// TIA Portal V17 export
// export: Created 2024-09-02T12:49:55.3240184Z, ExportSetting WithDefaults, DisplayName Totally Integrated Automation Portal, DisplayVersion V17, DisplayName TIA Portal Openness, DisplayVersion V17, DisplayName TIA Portal Version Control Interface, DisplayVersion V17, DisplayName STEP 7 Professional, DisplayVersion V17, DisplayName STEP 7 Safety, DisplayVersion V17, DisplayName WinCC Professional, DisplayVersion V17
FUNCTION "SysFC_AnzTrueDez" : Void   // FC128, LAD
TITLE = Count number of bits with value true / Anzahl Bits mit Wert true zaehlen
{ S7_Optimized_Access := 'TRUE' }
AUTHOR : OlegFuehrus
FAMILY : DIAG
NAME : DIAG
VERSION : 0.1
// stored: AutoNumber true, IsIECCheckEnabled false, SetENOAutomatically false, UDAEnableTagReadback false
   VAR_INPUT
      AnfangBits : Int;   // esrtes Bit zum zaehlen im Array / esrtes bit to count in array
      Anzahl : Int;   // Anzahl Bits zum überprüfen / Number of bits to check
      Daten : Variant;
   END_VAR
   VAR_OUTPUT
      AnzahlTrue : Int;   // Anzahl der Bits mit Wert True / Number of bits with value True
      NrTrue : Int;   // Nummer des ersten gefundenen Bits / Number of the first bit found
   END_VAR
   VAR_TEMP
      t_VKE0 : Bool;
      t_VKE1 : Bool;
      t_RetVal : Word;
      t_AnzahlElemente : UDInt;
      t_AnzahlTrue : Int;
      t_NrTrue : Int;
      t_PosNr : DInt;
      t_UDINT : UDInt;
      t_INT : Int;
      t_Counter : Int;
      t_StartCounter : Int;
      t_EndCounter : Int;
      t_Bool : Bool;
      t_Fehler : Bool;
      t_TypIO : Bool;
      t_DatenByte : Array[1..128] of Byte;
      t_DatenBool : Array[1..1024] of Bool;
   END_VAR
   VAR_TEMP   // added for the SCL form of the ladder/FBD networks
      _w1 : Bool;
   END_VAR
BEGIN

REGION Network 1: VKE0/1
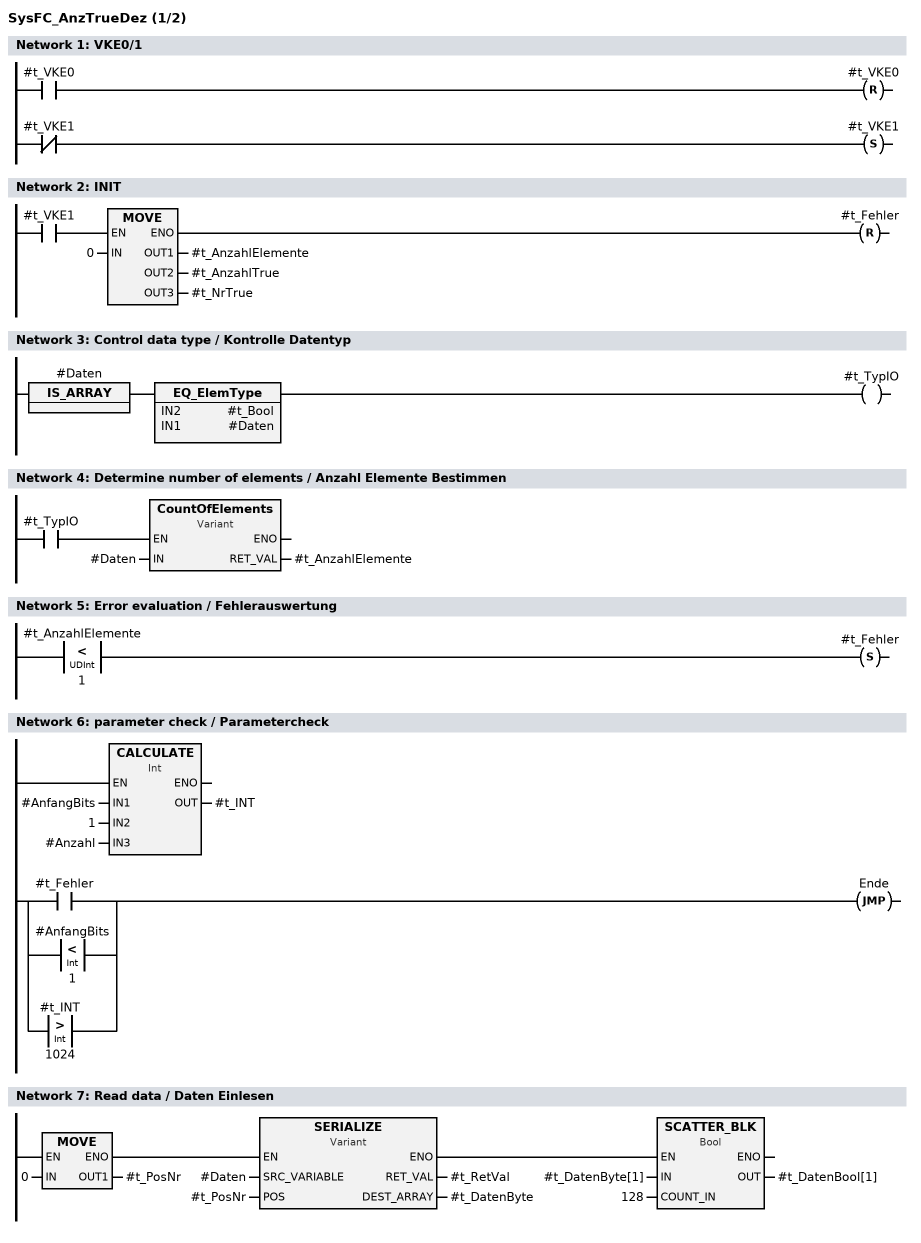
   RUNG wire#powerrail
      Contact( #t_VKE0 )
      R_Coil( #t_VKE0 )
   END_RUNG
   RUNG wire#powerrail
      I_Contact( #t_VKE1 )
      S_Coil( #t_VKE1 )
   END_RUNG
   // the same network as SCL:
   IF #t_VKE0 THEN #t_VKE0 := FALSE; END_IF;
   IF NOT #t_VKE1 THEN #t_VKE1 := TRUE; END_IF;
END_REGION

REGION Network 2: INIT
   RUNG wire#powerrail
      Contact( #t_VKE1 )
      Move(in := 0, out1 => #t_AnzahlElemente, out2 => #t_AnzahlTrue, out3 => #t_NrTrue)
      R_Coil( #t_Fehler )
   END_RUNG
   // the same network as SCL:
   IF #t_VKE1 THEN
       #t_AnzahlElemente := 0;
       #t_AnzahlTrue := 0;
       #t_NrTrue := 0;
       #t_Fehler := FALSE;
   END_IF;
END_REGION

REGION Network 3: Control data type / Kontrolle Datentyp
   // no SCL statement known for EQ_ElemType, IS_ARRAY: written as a call
   #t_TypIO := IS_ARRAY(#Daten) AND EQ_ElemType(in2 := #t_Bool, in1 := #Daten);
END_REGION

REGION Network 4: Determine number of elements / Anzahl Elemente Bestimmen
   // no SCL statement known for CountOfElements: written as a call
   IF #t_TypIO THEN #t_AnzahlElemente := CountOfElements(in := #Daten); END_IF;
END_REGION

REGION Network 5: Error evaluation / Fehlerauswertung
   RUNG wire#powerrail
      { S7_Templates := "SrcType := UDInt" } LT_Contact(in1 := #t_AnzahlElemente, in2 := 1)
      S_Coil( #t_Fehler )
   END_RUNG
   // the same network as SCL:
   IF #t_AnzahlElemente < 1 THEN #t_Fehler := TRUE; END_IF;
END_REGION

REGION Network 6: parameter check / Parametercheck
   RUNG wire#powerrail
      { S7_Templates := "SrcType := Int"; S7_Expression := "IN1-IN2+IN3" } Calculate(in1 := #AnfangBits, in2 := 1, in3 := #Anzahl, out => #t_INT)
   END_RUNG
   RUNG wire#powerrail
      Contact( #t_Fehler )
      wire#w1
      JumpCoil( Ende )
   END_RUNG
   RUNG wire#powerrail
      { S7_Templates := "SrcType := Int" } LT_Contact(in1 := #AnfangBits, in2 := 1)
   END_RUNG wire#w1
   RUNG wire#powerrail
      { S7_Templates := "SrcType := Int" } GT_Contact(in1 := #t_INT, in2 := 1024)
   END_RUNG wire#w1
   // the same network as SCL:
   #t_INT := #AnfangBits-1+#Anzahl;
   IF #t_Fehler OR (#AnfangBits < 1) OR (#t_INT > 1024) THEN GOTO Ende; END_IF;
END_REGION

REGION Network 7: Read data / Daten Einlesen
   RUNG wire#powerrail
      Move(in := 0, out1 => #t_PosNr)
      { S7_Templates := "var_type := Variant" } Serialize(SRC_VARIABLE := #Daten, POS := #t_PosNr, Ret_Val => #t_RetVal, DEST_ARRAY => #t_DatenByte)
      { S7_Templates := "[dest_type := Bool, src_type := Byte, count_type := UInt]" } SCATTER_BLK(IN := #t_DatenByte[1], COUNT_IN := 128, OUT => #t_DatenBool[1])
   END_RUNG
   // the same network as SCL:
   #t_PosNr := 0;
   #t_RetVal := Serialize(SRC_VARIABLE := #Daten, POS := #t_PosNr, DEST_ARRAY => #t_DatenByte, ENO => #_w1);
   IF #_w1 THEN SCATTER_BLK(IN := #t_DatenByte[1], COUNT_IN := 128, OUT => #t_DatenBool[1]); END_IF;
END_REGION

REGION Network 8 (SCL): Evaluate data / Daten Auswerten
   #t_Counter := int#0;
   #t_StartCounter := #AnfangBits;
   #t_EndCounter := #AnfangBits-1 + #Anzahl;

   FOR #t_Counter := #t_StartCounter TO #t_EndCounter DO
       IF #t_DatenBool[#t_Counter] = true THEN
           #t_AnzahlTrue := #t_AnzahlTrue + 1;

           IF #t_NrTrue = 0 THEN
               #t_NrTrue := #t_Counter;
           END_IF;

       END_IF;
   END_FOR;
END_REGION

REGION Network 9: Output / Ausgabe
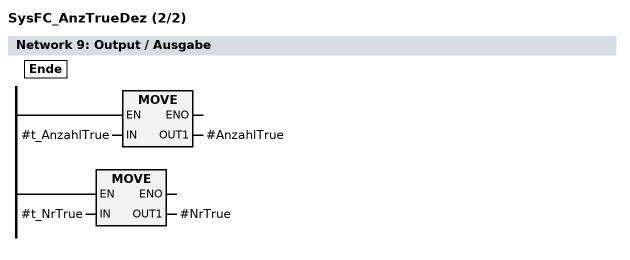
   Label( Ende )
   RUNG wire#powerrail
      Move(in := #t_AnzahlTrue, out1 => #AnzahlTrue)
   END_RUNG
   RUNG wire#powerrail
      Move(in := #t_NrTrue, out1 => #NrTrue)
   END_RUNG
   // the same network as SCL:
   Ende:
   #AnzahlTrue := #t_AnzahlTrue;
   #NrTrue := #t_NrTrue;
END_REGION
END_FUNCTION
